PROGRAM MAIN
VAR
	fbTimer : TON;
	i : INT;
END_VAR

fbTimer(IN:=TRUE, PT:=T#5S);
IF fbTimer.Q THEN
	i := i + 1;
	fbTimer(IN := FALSE);
END_IF

Test.nTest := i;

END_PROGRAM

(* stored: Version 1.1.0.1, ProductVersion 3.1.4024.12
   POU MAIN: Id {c11d7ff9-beaa-489d-8d9b-5b990bba7637}, SpecialFunc None *)
